# EPICS substitutions: ek9000App/Db/EL1034_mbbiDirect.substitutions
file EL1034.template
{       pattern
        {
                TERMINAL,

        }
        {
        }
}
